FUNCTION_BLOCK BasicSKILL_HMI (* Service Interface Function Block Type *)
  (* Standard: 61499-2 *)
  (* Version 0.0, 1/31/2024, midxav, template *)
  PACKAGE Main;
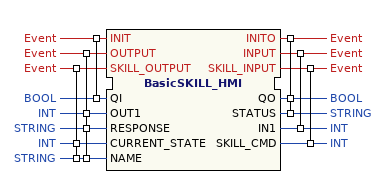
  EVENT_INPUT
    INIT WITH QI;
    OUTPUT WITH OUT1, RESPONSE, NAME;
    SKILL_OUTPUT WITH CURRENT_STATE, NAME;
  END_EVENT
  EVENT_OUTPUT
    INITO WITH QO, STATUS;
    INPUT WITH IN1;
    SKILL_INPUT WITH SKILL_CMD;
  END_EVENT
  VAR_INPUT
    QI : BOOL;
    OUT1 : INT;
    RESPONSE : STRING;
    CURRENT_STATE : INT;
    NAME : STRING;
  END_VAR
  VAR_OUTPUT
    QO : BOOL; (* Event Output Qualifier *)
    STATUS : STRING; (* Service Status *)
    IN1 : INT;
    SKILL_CMD : INT;
  END_VAR
  SERVICE /
    SEQUENCE 
    END_SEQUENCE
  END_SERVICE
END_FUNCTION_BLOCK
